FUNCTION_BLOCK CylinderService (* Message Exchange example (slide 47): SCylH / CylHServ - service-oriented cylinder, runs the physical round trip *)
  (* Standard: 61499-2; Description: Copyright (c) 2026 Meisterschulen am Ostbahnhof This program and the accompanying materials are made available under the terms of the Eclipse Public License 2.0 which is available at https://www.eclipse.org/legal/epl-2.0/ SPDX-License-Identifier: EPL-2.0 *)
  (* Version 1.0, 2026-09-03, Franz Höpfinger, Meisterschulen am Ostbahnhof, SoA implementation in function blocks (IEC 61499 primer course, Module 6, Valeriy Vyatkin, slide 47), SCylH/CylHServ role: uses full EVENT_HS_WSTRING (REQ/CNF/IND/RSP) - the only one of the four blocks that needs the mid-trip IND/RSP coordination (must pause after reaching the end position until the orchestrator confirms the drop) *)
  PACKAGE Meins::DesingPatterns::HandshakePattern;
  IMPORT Meins::DesingPatterns::HandshakePattern::const::MessageExchangeConst;
  (* Documentation:
  Service-oriented cylinder (SCylH/CylHServ in the "SoA implementation in function blocks" diagram, IEC 61499 primer course, Module 6, Valeriy Vyatkin, slide 47) - one of the four function blocks in the CylH message-exchange example (slides 42-46 for the message sequence chart this reconstructs).
   Uses EVENT_HS_WSTRING as a Socket (the only one of the four blocks that needs the full REQ/CNF/IND/RSP vocabulary, not a reduced variant): on REQ it starts the trip and fires an IND with RSP_CYL_STARTED; on the simulated AT_END sensor event it fires a second IND with RSP_CYL_END_POS and then waits for the matching RSP from CylinderOrchestrator before retracting - this is the one real synchronization point in the example: the physical cylinder must not start pulling back until the orchestrator confirms the workpiece was actually dropped. Once AT_START fires (pusher back home), it closes the transaction with CNF carrying RSP_CYL_TRIP_COMPLETE.
   Deliberate simplification vs. the full message-sequence chart: the low-level CYL.start/CYL.end/CYL.push/ CYL.pop sub-services from the MSC are not modelled as separate function blocks here - slide 47 itself treats SCylH/CylHServ as a single black box ("Interface to service-oriented cylinder"), so their internal push/pop/sensor choreography is folded into this one block's ECC instead, using AT_END/AT_START as the manually-fireable stand-ins for the physical sensors (same testing philosophy as EventDrivenCylinder.fbt in the Purely-Event-Driven pattern).
   See HandshakePattern.md in this folder, section "Die Quelle der 'push,100'-Notation", for the full write-up and the other three function blocks of this example (WorkpieceSensor, DropSinkService, CylinderOrchestrator).
  *)
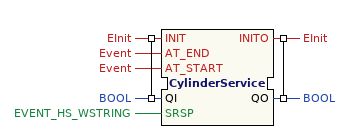
  EVENT_INPUT
    INIT : EInit WITH QI; (* Initialization Request *)
    AT_END; (* Simulated end-position sensor trigger: pusher reached the end position *)
    AT_START; (* Simulated start-position sensor trigger: pusher reached the start position again *)
  END_EVENT
  EVENT_OUTPUT
    INITO : EInit WITH QO; (* Initialization Confirm *)
  END_EVENT
  VAR_INPUT
    QI : BOOL; (* Input event qualifier *)
  END_VAR
  VAR_OUTPUT
    QO : BOOL; (* Output event qualifier *)
  END_VAR
  SOCKETS
    SRSP : adapter::types::bidirectional::Handshake::EVENT_HS_WSTRING; (* Service socket: receives REQ/RSP (+REQD/RSPD), emits CNF/IND (+CNFD/INDD) *)
  END_SOCKETS
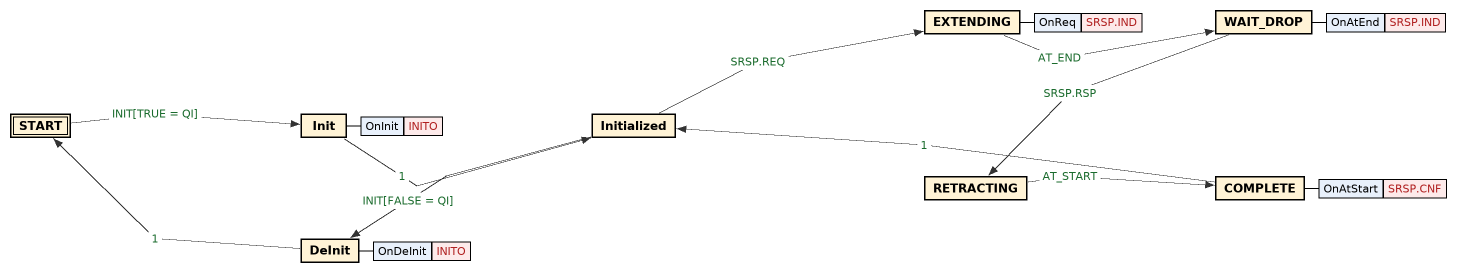
  EC_STATES
    START; (* Uninitialized *)
    Init : OnInit -> INITO; (* Initialization *)
    Initialized; (* Idle at start position, ready for a trip REQ *)
    DeInit : OnDeInit -> INITO; (* De-initialization *)
    EXTENDING : OnReq -> SRSP.IND; (* Trip started, push valve extending, waiting for AT_END *)
    WAIT_DROP : OnAtEnd -> SRSP.IND; (* Reached end position, reported it, waiting for the orchestrator's RSP before retracting *)
    RETRACTING; (* Drop acknowledged, push valve retracting / pop valve extending, waiting for AT_START *)
    COMPLETE : OnAtStart -> SRSP.CNF; (* Start position reached: close the transaction with CNF *)
  END_STATES
  EC_TRANSITIONS
    START TO Init := INIT[TRUE = QI];
    Init TO Initialized := 1;
    Initialized TO DeInit := INIT[FALSE = QI];
    DeInit TO START := 1;
    Initialized TO EXTENDING := SRSP.REQ;
    EXTENDING TO WAIT_DROP := AT_END;
    WAIT_DROP TO RETRACTING := SRSP.RSP;
    RETRACTING TO COMPLETE := AT_START;
    COMPLETE TO Initialized := 1;
  END_TRANSITIONS
  ALGORITHM OnInit IN ST: (* Initialize *)
QO := QI;
  END_ALGORITHM
  ALGORITHM OnDeInit IN ST: (* De-initialize *)
QO := FALSE;
  END_ALGORITHM
  ALGORITHM OnReq IN ST: (* Trip requested: begin extending, report the started status *)
SRSP.INDD := MessageExchangeConst::RSP_CYL_STARTED;
  END_ALGORITHM
  ALGORITHM OnAtEnd IN ST: (* End position reached: report it, then wait for the orchestrator's go-ahead *)
SRSP.INDD := MessageExchangeConst::RSP_CYL_END_POS;
  END_ALGORITHM
  ALGORITHM OnAtStart IN ST: (* Start position reached again: trip is complete *)
SRSP.CNFD := MessageExchangeConst::RSP_CYL_TRIP_COMPLETE;
  END_ALGORITHM
END_FUNCTION_BLOCK
